// TIA Portal V17 export
// export: Created 2025-03-07T09:16:31.8532208Z, ExportSetting WithDefaults, DisplayName Totally Integrated Automation Portal, DisplayVersion V17 Update 8, DisplayName TIA Portal Openness, DisplayVersion V17 Update 8, DisplayName TIA Portal Version Control Interface, DisplayVersion V17, DisplayName SINAMICS Startdrive Advanced, DisplayVersion V17 SP2, DisplayName SINAMICS Startdrive G110M, G120, G120C, G120D, G120P, G115D, DisplayVersion V17 SP2, DisplayName SINAMICS Startdrive G130, G150, S120, S150, SINAMICS MV, S210, DisplayVersion V17 SP2, DisplayName STEP 7 Professional, DisplayVersion V17 Update 8, DisplayName SINUMERIK ONE STEP 7 Toolbox, DisplayVersion V17 Update 12, DisplayName SINUMERIK 840D sl STEP 7 Toolbox, DisplayVersion V17 Update 12, DisplayName STEP 7 Safety, DisplayVersion V17 Update 6, DisplayName WinCC Advanced, DisplayVersion V17 Update 8
DATA_BLOCK "LBP_NC"   // DB10
TITLE = NC signals / Señales CN / NC-Signale
{ S7_Optimized_Access := 'FALSE'; DB_Accessible_From_OPC_UA := 'FALSE' }
AUTHOR : SINUMERIK
FAMILY : SINUMERIK_ONE
VERSION : 6.15
// Interface between user program and NC, contains signals from/to the NC, PLC and operating software. / Interfaz entre programa de usuario y CN, contiene señales desde/hacia CN, PLC y software operativo. / Schnittstelle zwischen Anwenderprogramm und NC, enthält Signale von/zu NC, PLC und Betriebssoftware.
// stored: AutoNumber false, DBAccessibleFromOPCUA false, DBAccessibleFromWebserver true, InstanceOfName LBP_typeNC, InstanceOfType UDT, IsOnlyStoredInLoadMemory false, IsWriteProtectedInAS false
"LBP_typeNC"
   // VAR RETAIN
   //    A_Disabl_Inp1 : Bool;
   //    A_Disabl_Inp2 : Bool;
   //    A_Disabl_Inp3 : Bool;
   //    A_Disabl_Inp4 : Bool;
   //    A_Disabl_Inp5 : Bool;
   //    A_Disabl_Inp6 : Bool;
   //    A_Disabl_Inp7 : Bool;
   //    A_Disabl_Inp8 : Bool;
   //    A_Set_Inp1 : Bool;
   //    A_Set_Inp2 : Bool;
   //    A_Set_Inp3 : Bool;
   //    A_Set_Inp4 : Bool;
   //    A_Set_Inp5 : Bool;
   //    A_Set_Inp6 : Bool;
   //    A_Set_Inp7 : Bool;
   //    A_Set_Inp8 : Bool;
   //    f0_f15 : Array[0..15] of Bool;
   //    A_Disabl_Out1 : Bool;
   //    A_Disabl_Out2 : Bool;
   //    A_Disabl_Out3 : Bool;
   //    A_Disabl_Out4 : Bool;
   //    A_Disabl_Out5 : Bool;
   //    A_Disabl_Out6 : Bool;
   //    A_Disabl_Out7 : Bool;
   //    A_Disabl_Out8 : Bool;
   //    A_OvMask_Out1 : Bool;
   //    A_OvMask_Out2 : Bool;
   //    A_OvMask_Out3 : Bool;
   //    A_OvMask_Out4 : Bool;
   //    A_OvMask_Out5 : Bool;
   //    A_OvMask_Out6 : Bool;
   //    A_OvMask_Out7 : Bool;
   //    A_OvMask_Out8 : Bool;
   //    A_Set_Out1 : Bool;
   //    A_Set_Out2 : Bool;
   //    A_Set_Out3 : Bool;
   //    A_Set_Out4 : Bool;
   //    A_Set_Out5 : Bool;
   //    A_Set_Out6 : Bool;
   //    A_Set_Out7 : Bool;
   //    A_Set_Out8 : Bool;
   //    A_InMask_Out1 : Bool;
   //    A_InMask_Out2 : Bool;
   //    A_InMask_Out3 : Bool;
   //    A_InMask_Out4 : Bool;
   //    A_InMask_Out5 : Bool;
   //    A_InMask_Out6 : Bool;
   //    A_InMask_Out7 : Bool;
   //    A_InMask_Out8 : Bool;
   //    MCP1AxisTbl : Array[1..22] of Byte;
   //    MCP1MaxAxis : Word;
   //    MCP2AxisTbl : Array[1..22] of Byte;
   //    MCP2MaxAxis : Word;
   //    f56_0 : Bool;
   //    A_EMERGENCY : Bool;
   //    A_EMERGENCY_Ackn : Bool;
   //    f56_3 : Bool;
   //    A_Keyswitch0 : Bool;
   //    A_Keyswitch1 : Bool;
   //    A_Keyswitch2 : Bool;
   //    A_Keyswitch3 : Bool;
   //    A_IncInModeGroup : Bool;
   //    f57_1 : Bool;
   //    f57_2 : Bool;
   //    A_PCshutdown : Bool;
   //    f57_4 : Bool;
   //    f57_5 : Bool;
   //    f57_6 : Bool;
   //    f57_7 : Bool;
   //    A_CA_DisableAutoMach : Bool;
   //    A_CA_DisableAutoTools : Bool;
   //    A_CA_DisableAutoWorkh : Bool;
   //    A_CA_DisableAutoWorkp : Bool;
   //    A_CA_DisableJogMach : Bool;
   //    A_CA_DisableJogTools : Bool;
   //    A_CA_DisableJogWorkh : Bool;
   //    A_CA_DisableJogWorkp : Bool;
   //    f59 : Byte;
   //    E_ActVal_In1 : Bool;
   //    E_ActVal_In2 : Bool;
   //    E_ActVal_In3 : Bool;
   //    E_ActVal_In4 : Bool;
   //    f60_4 : Bool;
   //    f60_5 : Bool;
   //    f60_6 : Bool;
   //    f60_7 : Bool;
   //    f61_f62 : Array[61..61] of Byte;
   //    E_Setpoint_Out1 : Bool;
   //    E_Setpoint_Out2 : Bool;
   //    E_Setpoint_Out3 : Bool;
   //    E_Setpoint_Out4 : Bool;
   //    E_Setpoint_Out5 : Bool;
   //    E_Setpoint_Out6 : Bool;
   //    E_Setpoint_Out7 : Bool;
   //    E_Setpoint_Out8 : Bool;
   //    f65_f67 : Array[65..66] of Byte;
   //    E_HW1_moved : Byte;
   //    E_HW2_moved : Byte;
   //    E_HW3_moved : Byte;
   //    E_CounterInchMetr : Byte;
   //    E_MCP1AxisValid : Bool;
   //    E_MCP1WCS : Bool;
   //    f72_2 : Bool;
   //    f72_3 : Bool;
   //    f72_4 : Bool;
   //    f72_5 : Bool;
   //    f72_6 : Bool;
   //    E_MCP1AxKeyDisp : Bool;
   //    E_MCP2AxisValid : Bool;
   //    E_MCP2WCS : Bool;
   //    f73_2 : Bool;
   //    f73_3 : Bool;
   //    f73_4 : Bool;
   //    f73_5 : Bool;
   //    f73_6 : Bool;
   //    E_MCP2AxKeyDisp : Bool;
   //    MCP1AxisFromHMI : Array[1..6] of Byte;
   //    MCP2AxisFromHMI : Array[1..6] of Byte;
   //    res86 : Word;
   //    res88 : Byte;
   //    res89 : Byte;
   //    epsToPlc : Byte;
   //    epsFromPlc : Byte;
   //    MpiDpOk : Bool;
   //    DpOk : Bool;
   //    PnOk : Bool;
   //    f92_3 : Bool;
   //    Disabl_AlarmMpiDp : Bool;
   //    Disabl_AlarmDp : Bool;
   //    Disabl_AlarmPn : Bool;
   //    f92_7 : Bool;
   //    E_CA_DisableAutoMach : Bool;
   //    E_CA_DisableAutoTools : Bool;
   //    E_CA_DisableAutoWorkh : Bool;
   //    E_CA_DisableAutoWorkp : Bool;
   //    E_CA_DisableJogMach : Bool;
   //    E_CA_DisableJogTools : Bool;
   //    E_CA_DisableJogWorkh : Bool;
   //    E_CA_DisableJogWorkp : Bool;
   //    E_MCP1LostPackageWarn : Bool;
   //    E_MCP2LostPackageWarn : Bool;
   //    E_HTLostPackageWarn : Bool;
   //    E_Op1KeyLostPackageWarn : Bool;
   //    E_Op2KeyLostPackageWarn : Bool;
   //    f94_5 : Bool;
   //    f94_6 : Bool;
   //    f94_7 : Bool;
   //    f95 : Byte;
   //    E_LanguageID : Byte;
   //    E_Chan_HW1_A : Bool;
   //    E_Chan_HW1_B : Bool;
   //    E_Chan_HW1_C : Bool;
   //    E_Chan_HW1_D : Bool;
   //    f97_4 : Bool;
   //    f97_5 : Bool;
   //    f97_6 : Bool;
   //    f97_7 : Bool;
   //    E_Chan_HW2_A : Bool;
   //    E_Chan_HW2_B : Bool;
   //    E_Chan_HW2_C : Bool;
   //    E_Chan_HW2_D : Bool;
   //    f98_4 : Bool;
   //    f98_5 : Bool;
   //    f98_6 : Bool;
   //    f98_7 : Bool;
   //    E_Chan_HW3_A : Bool;
   //    E_Chan_HW3_B : Bool;
   //    E_Chan_HW3_C : Bool;
   //    E_Chan_HW3_D : Bool;
   //    f99_4 : Bool;
   //    f99_5 : Bool;
   //    f99_6 : Bool;
   //    f99_7 : Bool;
   //    E_Ax_A_HW1 : Bool;
   //    E_Ax_B_HW1 : Bool;
   //    E_Ax_C_HW1 : Bool;
   //    E_Ax_D_HW1 : Bool;
   //    E_Ax_E_HW1 : Bool;
   //    E_CHW_sel1 : Bool;
   //    E_HW_sel1 : Bool;
   //    E_Mach_Ax1 : Bool;
   //    E_Ax_A_HW2 : Bool;
   //    E_Ax_B_HW2 : Bool;
   //    E_Ax_C_HW2 : Bool;
   //    E_Ax_D_HW2 : Bool;
   //    E_Ax_E_HW2 : Bool;
   //    E_CHW_sel2 : Bool;
   //    E_HW_sel2 : Bool;
   //    E_Mach_Ax2 : Bool;
   //    E_Ax_A_HW3 : Bool;
   //    E_Ax_B_HW3 : Bool;
   //    E_Ax_C_HW3 : Bool;
   //    E_Ax_D_HW3 : Bool;
   //    E_Ax_E_HW3 : Bool;
   //    E_CHW_sel3 : Bool;
   //    E_HW_sel3 : Bool;
   //    E_Mach_Ax3 : Bool;
   //    E_RemDiag : Bool;
   //    f103_1 : Bool;
   //    f103_2 : Bool;
   //    f103_3 : Bool;
   //    f103_4 : Bool;
   //    E_ATready : Bool;
   //    E_MMCTemp : Bool;
   //    E_MMCBatt : Bool;
   //    E_MCP1ready : Bool;
   //    E_MCP2ready : Bool;
   //    E_HTready : Bool;
   //    E_Op1KeyReady : Bool;
   //    E_Op2KeyReady : Bool;
   //    f104_5 : Bool;
   //    E_FirstOB1 : Bool;
   //    E_NCKready : Bool;
   //    E_CancelToolCmd : Bool;
   //    f105_1 : Bool;
   //    f105_2 : Bool;
   //    f105_3 : Bool;
   //    f105_4 : Bool;
   //    f105_5 : Bool;
   //    f105_6 : Bool;
   //    f105_7 : Bool;
   //    E_CollCheckOff : Bool;
   //    E_EMERGENCY : Bool;
   //    f106_2 : Bool;
   //    f106_3 : Bool;
   //    f106_4 : Bool;
   //    f106_5 : Bool;
   //    f106_6 : Bool;
   //    f106_7 : Bool;
   //    E_InspProbe1 : Bool;
   //    E_InspProbe2 : Bool;
   //    f107_2 : Bool;
   //    f107_3 : Bool;
   //    f107_4 : Bool;
   //    f107_5 : Bool;
   //    E_NCU_LinkActive : Bool;
   //    E_SystemInchDim : Bool;
   //    f108_0 : Bool;
   //    E_MMC2Ready : Bool;
   //    E_MMCMPIready : Bool;
   //    E_MMCBTSSready : Bool;
   //    f108_4 : Bool;
   //    E_DrivesInCylOp : Bool;
   //    E_611Dready : Bool;
   //    E_NCready : Bool;
   //    E_NCKalarm : Bool;
   //    f109_1 : Bool;
   //    f109_2 : Bool;
   //    f109_3 : Bool;
   //    A_PC_OSfault : Bool;
   //    E_HTempAlarm : Bool;
   //    E_ATempAlarm : Bool;
   //    E_BattAlarm : Bool;
   //    E_SWCamMinus : Array[0..31] of Bool;
   //    E_SWCamPlus : Array[0..31] of Bool;
   //    f118_f121 : Array[0..3] of Byte;
   //    A_Disabl_Inp9 : Bool;
   //    A_Disabl_Inp10 : Bool;
   //    A_Disabl_Inp11 : Bool;
   //    A_Disabl_Inp12 : Bool;
   //    A_Disabl_Inp13 : Bool;
   //    A_Disabl_Inp14 : Bool;
   //    A_Disabl_Inp15 : Bool;
   //    A_Disabl_Inp16 : Bool;
   //    A_Set_Inp9 : Bool;
   //    A_Set_Inp10 : Bool;
   //    A_Set_Inp11 : Bool;
   //    A_Set_Inp12 : Bool;
   //    A_Set_Inp13 : Bool;
   //    A_Set_Inp14 : Bool;
   //    A_Set_Inp15 : Bool;
   //    A_Set_Inp16 : Bool;
   //    A_Disabl_Inp17 : Bool;
   //    A_Disabl_Inp18 : Bool;
   //    A_Disabl_Inp19 : Bool;
   //    A_Disabl_Inp20 : Bool;
   //    A_Disabl_Inp21 : Bool;
   //    A_Disabl_Inp22 : Bool;
   //    A_Disabl_Inp23 : Bool;
   //    A_Disabl_Inp24 : Bool;
   //    A_Set_Inp17 : Bool;
   //    A_Set_Inp18 : Bool;
   //    A_Set_Inp19 : Bool;
   //    A_Set_Inp20 : Bool;
   //    A_Set_Inp21 : Bool;
   //    A_Set_Inp22 : Bool;
   //    A_Set_Inp23 : Bool;
   //    A_Set_Inp24 : Bool;
   //    A_Disabl_Inp25 : Bool;
   //    A_Disabl_Inp26 : Bool;
   //    A_Disabl_Inp27 : Bool;
   //    A_Disabl_Inp28 : Bool;
   //    A_Disabl_Inp29 : Bool;
   //    A_Disabl_Inp30 : Bool;
   //    A_Disabl_Inp31 : Bool;
   //    A_Disabl_Inp32 : Bool;
   //    A_Set_Inp25 : Bool;
   //    A_Set_Inp26 : Bool;
   //    A_Set_Inp27 : Bool;
   //    A_Set_Inp28 : Bool;
   //    A_Set_Inp29 : Bool;
   //    A_Set_Inp30 : Bool;
   //    A_Set_Inp31 : Bool;
   //    A_Set_Inp32 : Bool;
   //    A_Disabl_Inp33 : Bool;
   //    A_Disabl_Inp34 : Bool;
   //    A_Disabl_Inp35 : Bool;
   //    A_Disabl_Inp36 : Bool;
   //    A_Disabl_Inp37 : Bool;
   //    A_Disabl_Inp38 : Bool;
   //    A_Disabl_Inp39 : Bool;
   //    A_Disabl_Inp40 : Bool;
   //    A_Set_Inp33 : Bool;
   //    A_Set_Inp34 : Bool;
   //    A_Set_Inp35 : Bool;
   //    A_Set_Inp36 : Bool;
   //    A_Set_Inp37 : Bool;
   //    A_Set_Inp38 : Bool;
   //    A_Set_Inp39 : Bool;
   //    A_Set_Inp40 : Bool;
   //    A_Disabl_Out9 : Bool;
   //    A_Disabl_Out10 : Bool;
   //    A_Disabl_Out11 : Bool;
   //    A_Disabl_Out12 : Bool;
   //    A_Disabl_Out13 : Bool;
   //    A_Disabl_Out14 : Bool;
   //    A_Disabl_Out15 : Bool;
   //    A_Disabl_Out16 : Bool;
   //    A_OvMask_Out9 : Bool;
   //    A_OvMask_Out10 : Bool;
   //    A_OvMask_Out11 : Bool;
   //    A_OvMask_Out12 : Bool;
   //    A_OvMask_Out13 : Bool;
   //    A_OvMask_Out14 : Bool;
   //    A_OvMask_Out15 : Bool;
   //    A_OvMask_Out16 : Bool;
   //    A_Set_Out9 : Bool;
   //    A_Set_Out10 : Bool;
   //    A_Set_Out11 : Bool;
   //    A_Set_Out12 : Bool;
   //    A_Set_Out13 : Bool;
   //    A_Set_Out14 : Bool;
   //    A_Set_Out15 : Bool;
   //    A_Set_Out16 : Bool;
   //    A_InMask_Out9 : Bool;
   //    A_InMask_Out10 : Bool;
   //    A_InMask_Out11 : Bool;
   //    A_InMask_Out12 : Bool;
   //    A_InMask_Out13 : Bool;
   //    A_InMask_Out14 : Bool;
   //    A_InMask_Out15 : Bool;
   //    A_InMask_Out16 : Bool;
   //    A_Disabl_Out17 : Bool;
   //    A_Disabl_Out18 : Bool;
   //    A_Disabl_Out19 : Bool;
   //    A_Disabl_Out20 : Bool;
   //    A_Disabl_Out21 : Bool;
   //    A_Disabl_Out22 : Bool;
   //    A_Disabl_Out23 : Bool;
   //    A_Disabl_Out24 : Bool;
   //    A_OvMask_Out17 : Bool;
   //    A_OvMask_Out18 : Bool;
   //    A_OvMask_Out19 : Bool;
   //    A_OvMask_Out20 : Bool;
   //    A_OvMask_Out21 : Bool;
   //    A_OvMask_Out22 : Bool;
   //    A_OvMask_Out23 : Bool;
   //    A_OvMask_Out24 : Bool;
   //    A_Set_Out17 : Bool;
   //    A_Set_Out18 : Bool;
   //    A_Set_Out19 : Bool;
   //    A_Set_Out20 : Bool;
   //    A_Set_Out21 : Bool;
   //    A_Set_Out22 : Bool;
   //    A_Set_Out23 : Bool;
   //    A_Set_Out24 : Bool;
   //    A_InMask_Out17 : Bool;
   //    A_InMask_Out18 : Bool;
   //    A_InMask_Out19 : Bool;
   //    A_InMask_Out20 : Bool;
   //    A_InMask_Out21 : Bool;
   //    A_InMask_Out22 : Bool;
   //    A_InMask_Out23 : Bool;
   //    A_InMask_Out24 : Bool;
   //    A_Disabl_Out25 : Bool;
   //    A_Disabl_Out26 : Bool;
   //    A_Disabl_Out27 : Bool;
   //    A_Disabl_Out28 : Bool;
   //    A_Disabl_Out29 : Bool;
   //    A_Disabl_Out30 : Bool;
   //    A_Disabl_Out31 : Bool;
   //    A_Disabl_Out32 : Bool;
   //    A_OvMask_Out25 : Bool;
   //    A_OvMask_Out26 : Bool;
   //    A_OvMask_Out27 : Bool;
   //    A_OvMask_Out28 : Bool;
   //    A_OvMask_Out29 : Bool;
   //    A_OvMask_Out30 : Bool;
   //    A_OvMask_Out31 : Bool;
   //    A_OvMask_Out32 : Bool;
   //    A_Set_Out25 : Bool;
   //    A_Set_Out26 : Bool;
   //    A_Set_Out27 : Bool;
   //    A_Set_Out28 : Bool;
   //    A_Set_Out29 : Bool;
   //    A_Set_Out30 : Bool;
   //    A_Set_Out31 : Bool;
   //    A_Set_Out32 : Bool;
   //    A_InMask_Out25 : Bool;
   //    A_InMask_Out26 : Bool;
   //    A_InMask_Out27 : Bool;
   //    A_InMask_Out28 : Bool;
   //    A_InMask_Out29 : Bool;
   //    A_InMask_Out30 : Bool;
   //    A_InMask_Out31 : Bool;
   //    A_InMask_Out32 : Bool;
   //    A_Disabl_Out33 : Bool;
   //    A_Disabl_Out34 : Bool;
   //    A_Disabl_Out35 : Bool;
   //    A_Disabl_Out36 : Bool;
   //    A_Disabl_Out37 : Bool;
   //    A_Disabl_Out38 : Bool;
   //    A_Disabl_Out39 : Bool;
   //    A_Disabl_Out40 : Bool;
   //    A_OvMask_Out33 : Bool;
   //    A_OvMask_Out34 : Bool;
   //    A_OvMask_Out35 : Bool;
   //    A_OvMask_Out36 : Bool;
   //    A_OvMask_Out37 : Bool;
   //    A_OvMask_Out38 : Bool;
   //    A_OvMask_Out39 : Bool;
   //    A_OvMask_Out40 : Bool;
   //    A_Set_Out33 : Bool;
   //    A_Set_Out34 : Bool;
   //    A_Set_Out35 : Bool;
   //    A_Set_Out36 : Bool;
   //    A_Set_Out37 : Bool;
   //    A_Set_Out38 : Bool;
   //    A_Set_Out39 : Bool;
   //    A_Set_Out40 : Bool;
   //    A_InMask_Out33 : Bool;
   //    A_InMask_Out34 : Bool;
   //    A_InMask_Out35 : Bool;
   //    A_InMask_Out36 : Bool;
   //    A_InMask_Out37 : Bool;
   //    A_InMask_Out38 : Bool;
   //    A_InMask_Out39 : Bool;
   //    A_InMask_Out40 : Bool;
   //    A_Disabl_anaIn1 : Bool;
   //    A_Disabl_anaIn2 : Bool;
   //    A_Disabl_anaIn3 : Bool;
   //    A_Disabl_anaIn4 : Bool;
   //    A_Disabl_anaIn5 : Bool;
   //    A_Disabl_anaIn6 : Bool;
   //    A_Disabl_anaIn7 : Bool;
   //    A_Disabl_anaIn8 : Bool;
   //    A_InMask_anaIn1 : Bool;
   //    A_InMask_anaIn2 : Bool;
   //    A_InMask_anaIn3 : Bool;
   //    A_InMask_anaIn4 : Bool;
   //    A_InMask_anaIn5 : Bool;
   //    A_InMask_anaIn6 : Bool;
   //    A_InMask_anaIn7 : Bool;
   //    A_InMask_anaIn8 : Bool;
   //    A_Setval_anaIn1 : Word;
   //    A_Setval_anaIn2 : Word;
   //    A_Setval_anaIn3 : Word;
   //    A_Setval_anaIn4 : Word;
   //    A_Setval_anaIn5 : Word;
   //    A_Setval_anaIn6 : Word;
   //    A_Setval_anaIn7 : Word;
   //    A_Setval_anaIn8 : Word;
   //    f164_f165 : Int;
   //    A_OvMask_anaOut1 : Bool;
   //    A_OvMask_anaOut2 : Bool;
   //    A_OvMask_anaOut3 : Bool;
   //    A_OvMask_anaOut4 : Bool;
   //    A_OvMask_anaOut5 : Bool;
   //    A_OvMask_anaOut6 : Bool;
   //    A_OvMask_anaOut7 : Bool;
   //    A_OvMask_anaOut8 : Bool;
   //    A_InMask_anaOut1 : Bool;
   //    A_InMask_anaOut2 : Bool;
   //    A_InMask_anaOut3 : Bool;
   //    A_InMask_anaOut4 : Bool;
   //    A_InMask_anaOut5 : Bool;
   //    A_InMask_anaOut6 : Bool;
   //    A_InMask_anaOut7 : Bool;
   //    A_InMask_anaOut8 : Bool;
   //    A_Disabl_anaOut1 : Bool;
   //    A_Disabl_anaOut2 : Bool;
   //    A_Disabl_anaOut3 : Bool;
   //    A_Disabl_anaOut4 : Bool;
   //    A_Disabl_anaOut5 : Bool;
   //    A_Disabl_anaOut6 : Bool;
   //    A_Disabl_anaOut7 : Bool;
   //    A_Disabl_anaOut8 : Bool;
   //    f169 : Byte;
   //    A_Setval_anaOut1 : Word;
   //    A_Setval_anaOut2 : Word;
   //    A_Setval_anaOut3 : Word;
   //    A_Setval_anaOut4 : Word;
   //    A_Setval_anaOut5 : Word;
   //    A_Setval_anaOut6 : Word;
   //    A_Setval_anaOut7 : Word;
   //    A_Setval_anaOut8 : Word;
   //    E_ActVal_In9 : Bool;
   //    E_ActVal_In10 : Bool;
   //    E_ActVal_In11 : Bool;
   //    E_ActVal_In12 : Bool;
   //    E_ActVal_In13 : Bool;
   //    E_ActVal_In14 : Bool;
   //    E_ActVal_In15 : Bool;
   //    E_ActVal_In16 : Bool;
   //    E_ActVal_In17 : Bool;
   //    E_ActVal_In18 : Bool;
   //    E_ActVal_In19 : Bool;
   //    E_ActVal_In20 : Bool;
   //    E_ActVal_In21 : Bool;
   //    E_ActVal_In22 : Bool;
   //    E_ActVal_In23 : Bool;
   //    E_ActVal_In24 : Bool;
   //    E_ActVal_In25 : Bool;
   //    E_ActVal_In26 : Bool;
   //    E_ActVal_In27 : Bool;
   //    E_ActVal_In28 : Bool;
   //    E_ActVal_In29 : Bool;
   //    E_ActVal_In30 : Bool;
   //    E_ActVal_In31 : Bool;
   //    E_ActVal_In32 : Bool;
   //    E_ActVal_In33 : Bool;
   //    E_ActVal_In34 : Bool;
   //    E_ActVal_In35 : Bool;
   //    E_ActVal_In36 : Bool;
   //    E_ActVal_In37 : Bool;
   //    E_ActVal_In38 : Bool;
   //    E_ActVal_In39 : Bool;
   //    E_ActVal_In40 : Bool;
   //    E_Setpoint_Out9 : Bool;
   //    E_Setpoint_Out10 : Bool;
   //    E_Setpoint_Out11 : Bool;
   //    E_Setpoint_Out12 : Bool;
   //    E_Setpoint_Out13 : Bool;
   //    E_Setpoint_Out14 : Bool;
   //    E_Setpoint_Out15 : Bool;
   //    E_Setpoint_Out16 : Bool;
   //    E_Setpoint_Out17 : Bool;
   //    E_Setpoint_Out18 : Bool;
   //    E_Setpoint_Out19 : Bool;
   //    E_Setpoint_Out20 : Bool;
   //    E_Setpoint_Out21 : Bool;
   //    E_Setpoint_Out22 : Bool;
   //    E_Setpoint_Out23 : Bool;
   //    E_Setpoint_Out24 : Bool;
   //    E_Setpoint_Out25 : Bool;
   //    E_Setpoint_Out26 : Bool;
   //    E_Setpoint_Out27 : Bool;
   //    E_Setpoint_Out28 : Bool;
   //    E_Setpoint_Out29 : Bool;
   //    E_Setpoint_Out30 : Bool;
   //    E_Setpoint_Out31 : Bool;
   //    E_Setpoint_Out32 : Bool;
   //    E_Setpoint_Out33 : Bool;
   //    E_Setpoint_Out34 : Bool;
   //    E_Setpoint_Out35 : Bool;
   //    E_Setpoint_Out36 : Bool;
   //    E_Setpoint_Out37 : Bool;
   //    E_Setpoint_Out38 : Bool;
   //    E_Setpoint_Out39 : Bool;
   //    E_Setpoint_Out40 : Bool;
   //    E_ActVal_anaIn1 : Word;
   //    E_ActVal_anaIn2 : Word;
   //    E_ActVal_anaIn3 : Word;
   //    E_ActVal_anaIn4 : Word;
   //    E_ActVal_anaIn5 : Word;
   //    E_ActVal_anaIn6 : Word;
   //    E_ActVal_anaIn7 : Word;
   //    E_ActVal_anaIn8 : Word;
   //    E_Setval_anaOut1 : Word;
   //    E_Setval_anaOut2 : Word;
   //    E_Setval_anaOut3 : Word;
   //    E_Setval_anaOut4 : Word;
   //    E_Setval_anaOut5 : Word;
   //    E_Setval_anaOut6 : Word;
   //    E_Setval_anaOut7 : Word;
   //    E_Setval_anaOut8 : Word;
   //    E_CollCheck : Array[0..7] of Byte;
   //    A_CollCheck : Array[0..7] of Byte;
   //    E_HW4_moved : Byte;
   //    E_HW5_moved : Byte;
   //    E_HW6_moved : Byte;
   //    E_EHW1_stands : Bool;
   //    E_EHW2_stands : Bool;
   //    E_EHW3_stands : Bool;
   //    E_EHW4_stands : Bool;
   //    E_EHW5_stands : Bool;
   //    E_EHW6_stands : Bool;
   //    f245_6 : Bool;
   //    f245_7 : Bool;
   //    E_HMI_HW1Active : Bool;
   //    E_HMI_HW2Active : Bool;
   //    E_HMI_HW3Active : Bool;
   //    E_HMI_HW4Active : Bool;
   //    E_HMI_HW5Active : Bool;
   //    E_HMI_HW6Active : Bool;
   //    f246_6 : Bool;
   //    f246_7 : Bool;
   //    f247 : Byte;
   //    A_RobotStatus : Array[0..7] of Byte;
   //    E_RobotControl : Array[0..7] of Byte;
   // END_VAR
BEGIN
END_DATA_BLOCK
